(* PLC project AKS_v2.project, Prosoft-Systems Ltd. Astra.IDE Astra.IDE_V1.7.2.1 *)
(* stored: creationDateTime 2025-07-24T10:35:59.4336606, modificationDateTime 2025-07-24T08:15:04.4598718 *)

{attribute 'object_name' := 'AI__1'}
PROGRAM Generated_2025_07_28
  VAR
    DI_DI : FB_DI;
    A : BOOL;
    B : BOOL;
    DI_DI : FB_DI;
    A : BOOL;
    B : BOOL;
    DI_DI : FB_DI;
    A : BOOL;
    B : BOOL;
    DI_DI : FB_DI;
    A : BOOL;
    B : BOOL;
    DI_DI : FB_DI;
    A : BOOL;
    B : BOOL;
  END_VAR

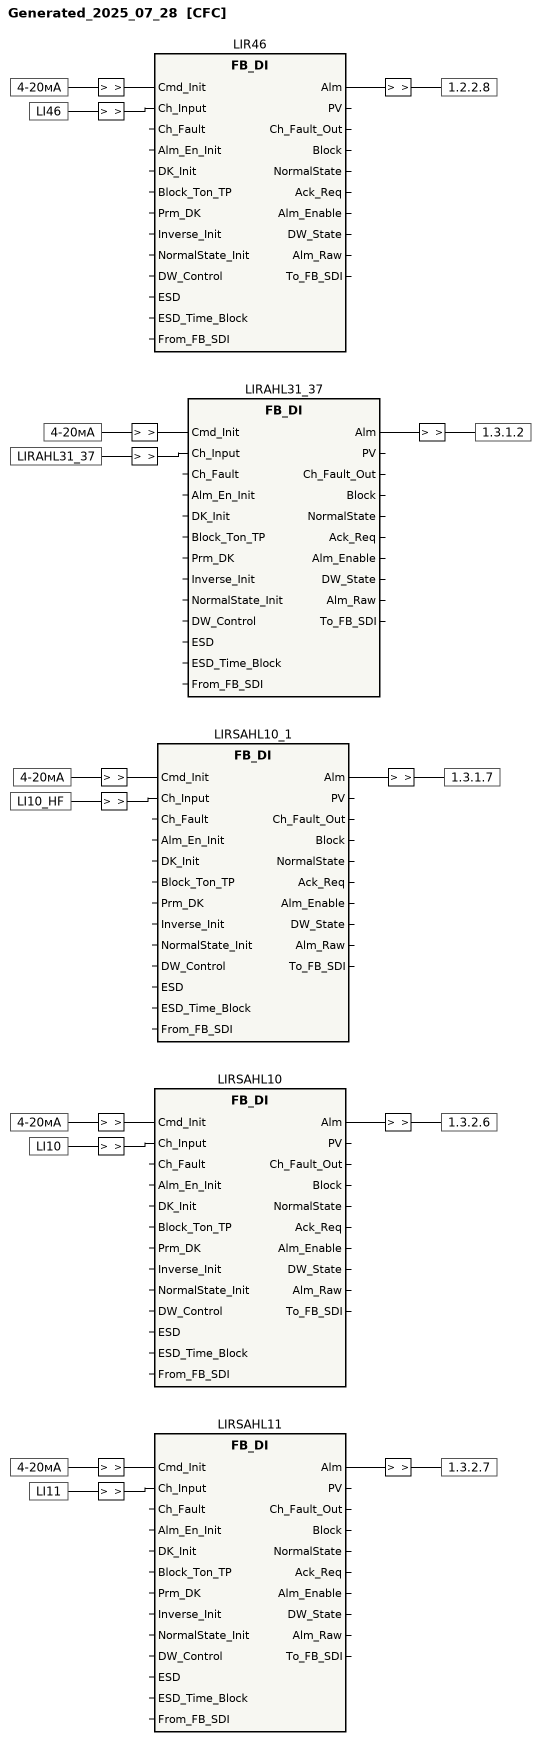
(* CFC diagram, written out as Structured Text *)
1.2.2.8 := LIR46.Alm;
1.3.1.2 := LIRAHL31_37.Alm;
1.3.1.7 := LIRSAHL10_1.Alm;
1.3.2.6 := LIRSAHL10.Alm;
1.3.2.7 := LIRSAHL11.Alm;
LIR46(Cmd_Init := 4-20мA, Ch_Input := LI46);
LIRAHL31_37(Cmd_Init := 4-20мA, Ch_Input := LIRAHL31_37);
LIRSAHL10_1(Cmd_Init := 4-20мA, Ch_Input := LI10_HF);
LIRSAHL10(Cmd_Init := 4-20мA, Ch_Input := LI10);
LIRSAHL11(Cmd_Init := 4-20мA, Ch_Input := LI11);
END_PROGRAM
